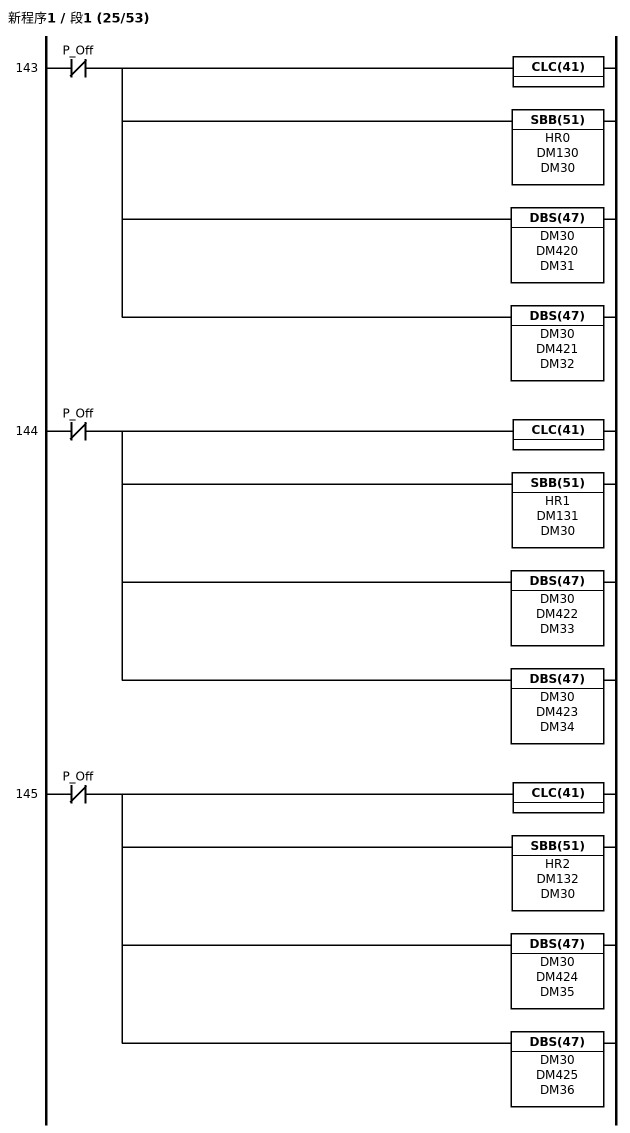
; [picture p24: 新程序1 / 段1, rungs 143-145]
; rung 143
LDNOT P_Off
CLC(41)
SBB(51) HR0 DM130 DM30
DBS(47) DM30 DM420 DM31
DBS(47) DM30 DM421 DM32
; rung 144
LDNOT P_Off
CLC(41)
SBB(51) HR1 DM131 DM30
DBS(47) DM30 DM422 DM33
DBS(47) DM30 DM423 DM34
; rung 145
LDNOT P_Off
CLC(41)
SBB(51) HR2 DM132 DM30
DBS(47) DM30 DM424 DM35
DBS(47) DM30 DM425 DM36

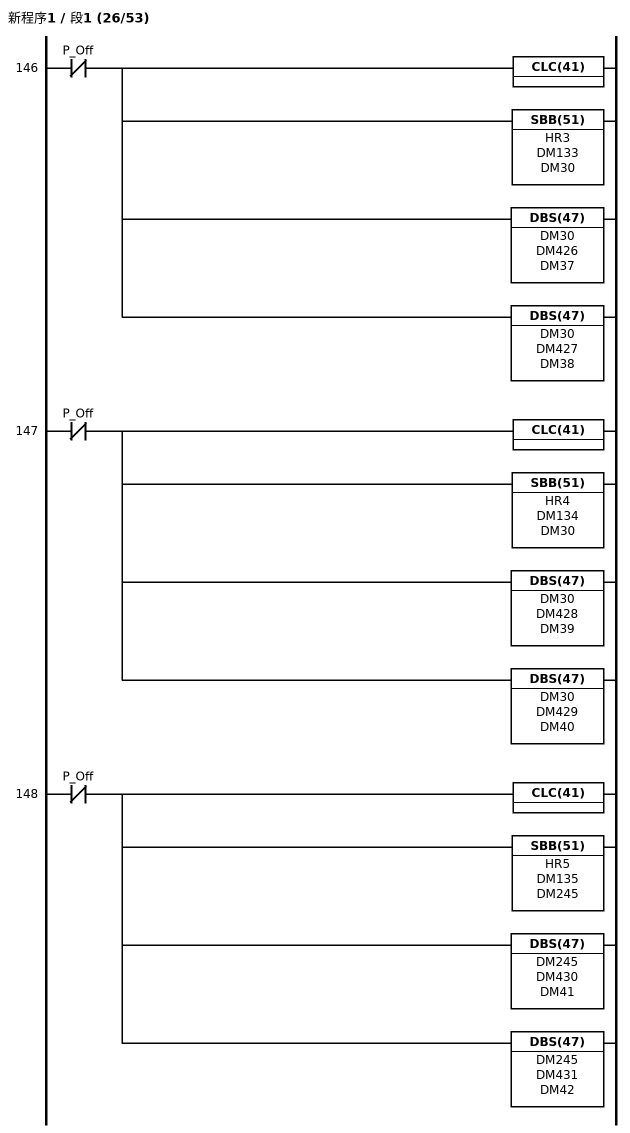
; rung 146
LDNOT P_Off
CLC(41)
SBB(51) HR3 DM133 DM30
DBS(47) DM30 DM426 DM37
DBS(47) DM30 DM427 DM38
; rung 147
LDNOT P_Off
CLC(41)
SBB(51) HR4 DM134 DM30
DBS(47) DM30 DM428 DM39
DBS(47) DM30 DM429 DM40
; rung 148
LDNOT P_Off
CLC(41)
SBB(51) HR5 DM135 DM245
DBS(47) DM245 DM430 DM41
DBS(47) DM245 DM431 DM42

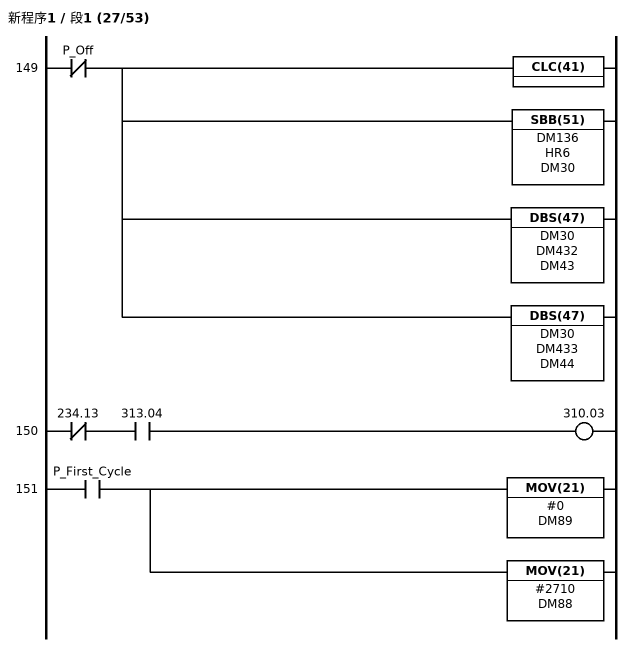
; rung 149
LDNOT P_Off
CLC(41)
SBB(51) DM136 HR6 DM30
DBS(47) DM30 DM432 DM43
DBS(47) DM30 DM433 DM44
; rung 150
LDNOT 234.13
AND 313.04
OUT 310.03
; rung 151
LD P_First_Cycle
MOV(21) #0 DM89
MOV(21) #2710 DM88

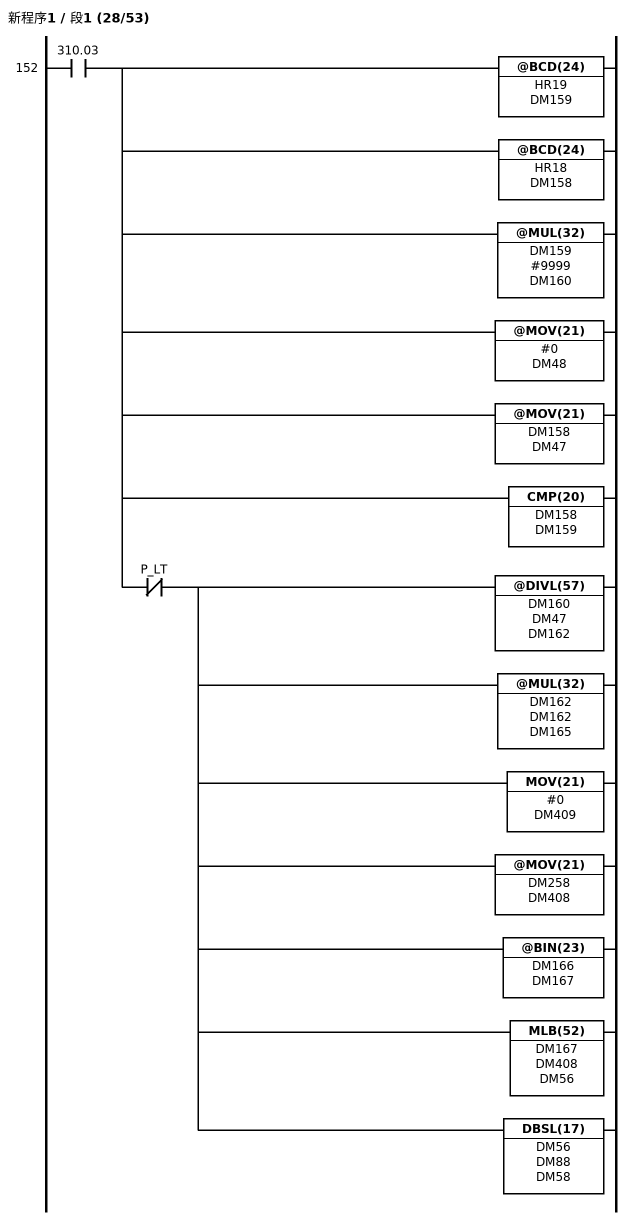
; rung 152
LD 310.03
@BCD(24) HR19 DM159
@BCD(24) HR18 DM158
@MUL(32) DM159 #9999 DM160
@MOV(21) #0 DM48
@MOV(21) DM158 DM47
CMP(20) DM158 DM159
ANDNOT P_LT
@DIVL(57) DM160 DM47 DM162
@MUL(32) DM162 DM162 DM165
MOV(21) #0 DM409
@MOV(21) DM258 DM408
@BIN(23) DM166 DM167
MLB(52) DM167 DM408 DM56
DBSL(17) DM56 DM88 DM58

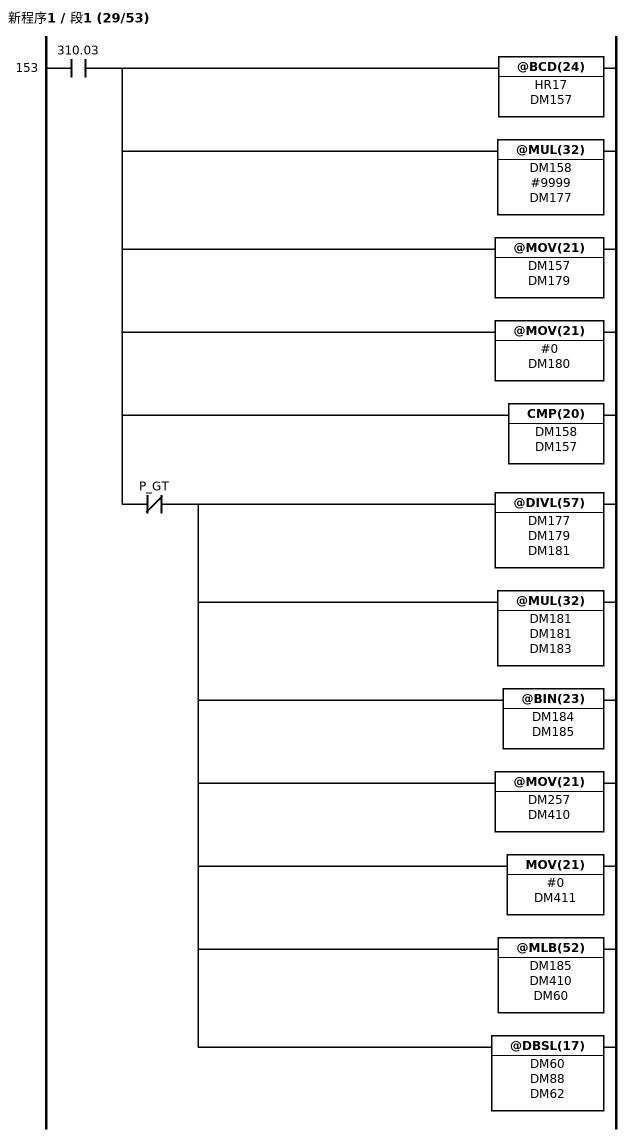
; rung 153
LD 310.03
@BCD(24) HR17 DM157
@MUL(32) DM158 #9999 DM177
@MOV(21) DM157 DM179
@MOV(21) #0 DM180
CMP(20) DM158 DM157
ANDNOT P_GT
@DIVL(57) DM177 DM179 DM181
@MUL(32) DM181 DM181 DM183
@BIN(23) DM184 DM185
@MOV(21) DM257 DM410
MOV(21) #0 DM411
@MLB(52) DM185 DM410 DM60
@DBSL(17) DM60 DM88 DM62

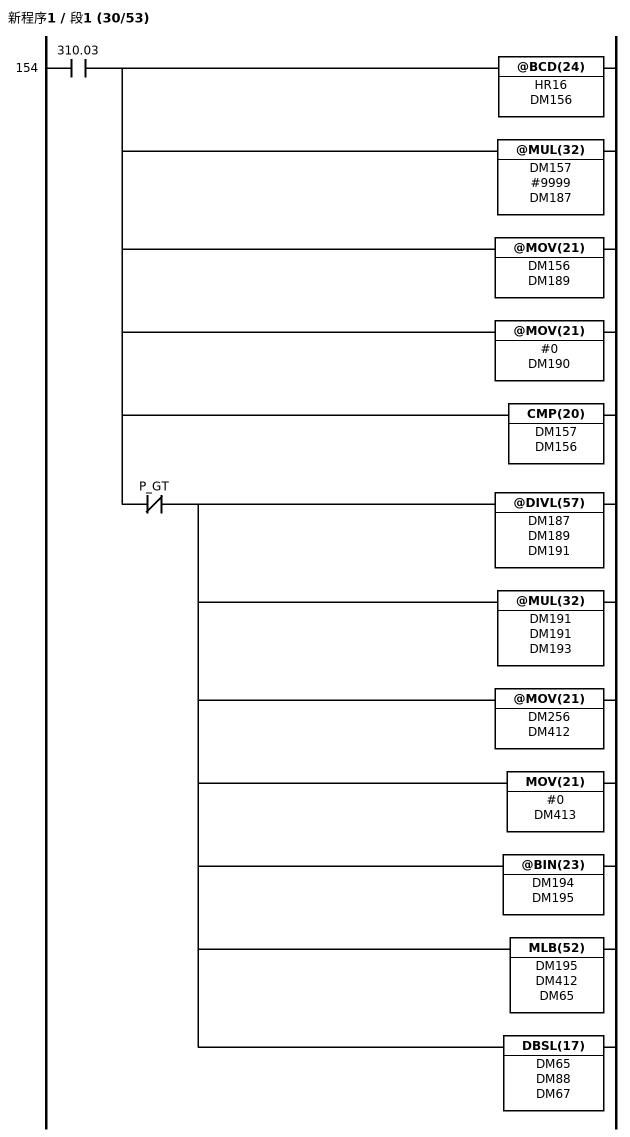
; rung 154
LD 310.03
@BCD(24) HR16 DM156
@MUL(32) DM157 #9999 DM187
@MOV(21) DM156 DM189
@MOV(21) #0 DM190
CMP(20) DM157 DM156
ANDNOT P_GT
@DIVL(57) DM187 DM189 DM191
@MUL(32) DM191 DM191 DM193
@MOV(21) DM256 DM412
MOV(21) #0 DM413
@BIN(23) DM194 DM195
MLB(52) DM195 DM412 DM65
DBSL(17) DM65 DM88 DM67

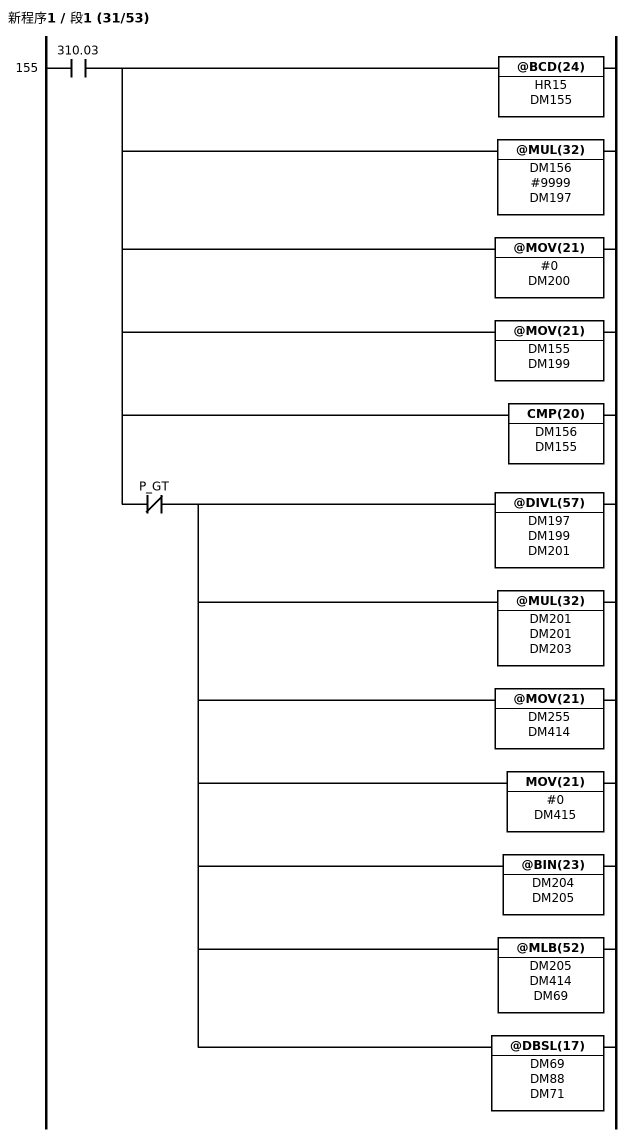
; rung 155
LD 310.03
@BCD(24) HR15 DM155
@MUL(32) DM156 #9999 DM197
@MOV(21) #0 DM200
@MOV(21) DM155 DM199
CMP(20) DM156 DM155
ANDNOT P_GT
@DIVL(57) DM197 DM199 DM201
@MUL(32) DM201 DM201 DM203
@MOV(21) DM255 DM414
MOV(21) #0 DM415
@BIN(23) DM204 DM205
@MLB(52) DM205 DM414 DM69
@DBSL(17) DM69 DM88 DM71

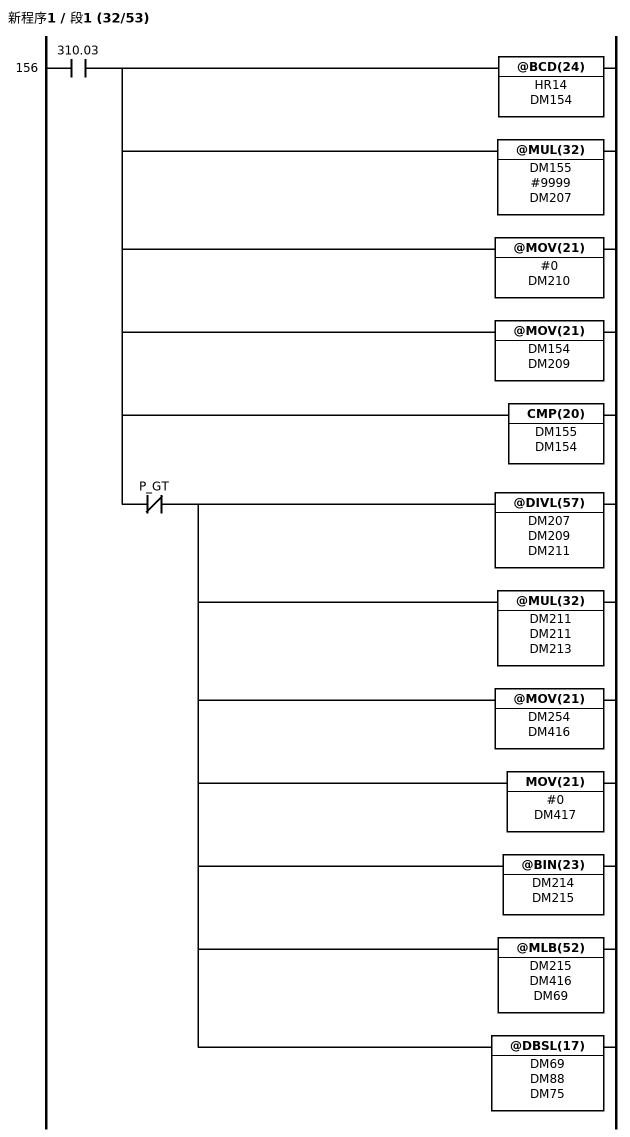
; rung 156
LD 310.03
@BCD(24) HR14 DM154
@MUL(32) DM155 #9999 DM207
@MOV(21) #0 DM210
@MOV(21) DM154 DM209
CMP(20) DM155 DM154
ANDNOT P_GT
@DIVL(57) DM207 DM209 DM211
@MUL(32) DM211 DM211 DM213
@MOV(21) DM254 DM416
MOV(21) #0 DM417
@BIN(23) DM214 DM215
@MLB(52) DM215 DM416 DM69
@DBSL(17) DM69 DM88 DM75

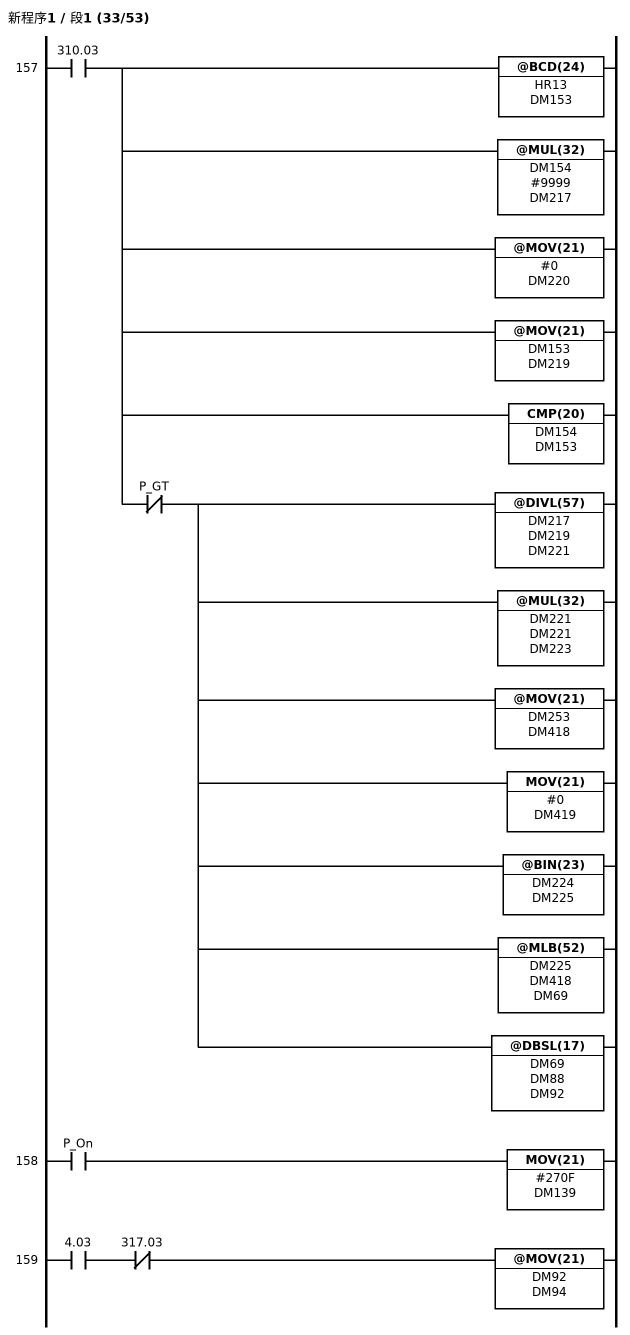
; rung 157
LD 310.03
@BCD(24) HR13 DM153
@MUL(32) DM154 #9999 DM217
@MOV(21) #0 DM220
@MOV(21) DM153 DM219
CMP(20) DM154 DM153
ANDNOT P_GT
@DIVL(57) DM217 DM219 DM221
@MUL(32) DM221 DM221 DM223
@MOV(21) DM253 DM418
MOV(21) #0 DM419
@BIN(23) DM224 DM225
@MLB(52) DM225 DM418 DM69
@DBSL(17) DM69 DM88 DM92
; rung 158
LD P_On
MOV(21) #270F DM139
; rung 159
LD 4.03
ANDNOT 317.03
@MOV(21) DM92 DM94

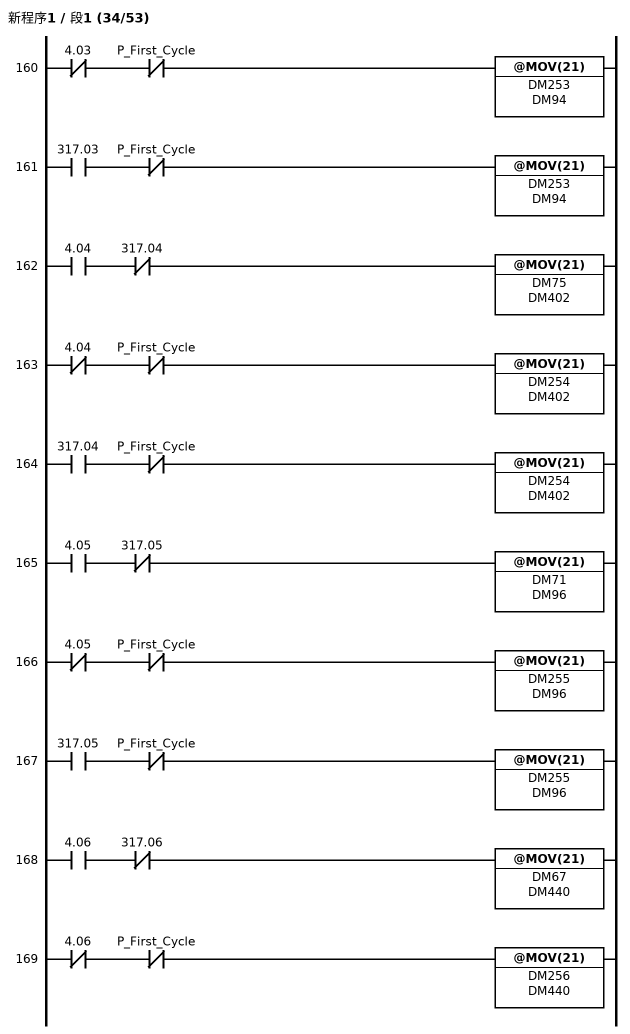
; rung 160
LDNOT 4.03
ANDNOT P_First_Cycle
@MOV(21) DM253 DM94
; rung 161
LD 317.03
ANDNOT P_First_Cycle
@MOV(21) DM253 DM94
; rung 162
LD 4.04
ANDNOT 317.04
@MOV(21) DM75 DM402
; rung 163
LDNOT 4.04
ANDNOT P_First_Cycle
@MOV(21) DM254 DM402
; rung 164
LD 317.04
ANDNOT P_First_Cycle
@MOV(21) DM254 DM402
; rung 165
LD 4.05
ANDNOT 317.05
@MOV(21) DM71 DM96
; rung 166
LDNOT 4.05
ANDNOT P_First_Cycle
@MOV(21) DM255 DM96
; rung 167
LD 317.05
ANDNOT P_First_Cycle
@MOV(21) DM255 DM96
; rung 168
LD 4.06
ANDNOT 317.06
@MOV(21) DM67 DM440
; rung 169
LDNOT 4.06
ANDNOT P_First_Cycle
@MOV(21) DM256 DM440

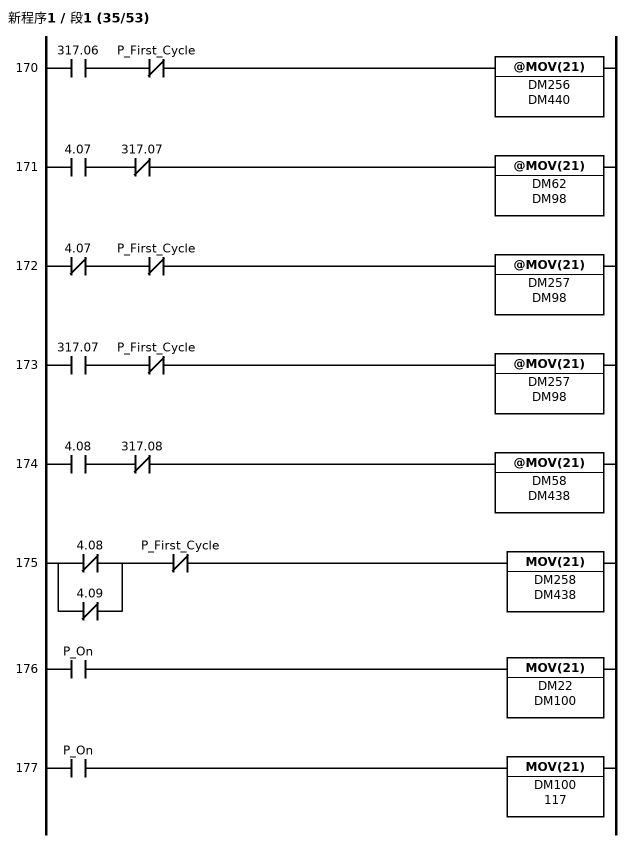
; rung 170
LD 317.06
ANDNOT P_First_Cycle
@MOV(21) DM256 DM440
; rung 171
LD 4.07
ANDNOT 317.07
@MOV(21) DM62 DM98
; rung 172
LDNOT 4.07
ANDNOT P_First_Cycle
@MOV(21) DM257 DM98
; rung 173
LD 317.07
ANDNOT P_First_Cycle
@MOV(21) DM257 DM98
; rung 174
LD 4.08
ANDNOT 317.08
@MOV(21) DM58 DM438
; rung 175
LDNOT 4.08
ORNOT 4.09
ANDNOT P_First_Cycle
MOV(21) DM258 DM438
; rung 176
LD P_On
MOV(21) DM22 DM100
; rung 177
LD P_On
MOV(21) DM100 117

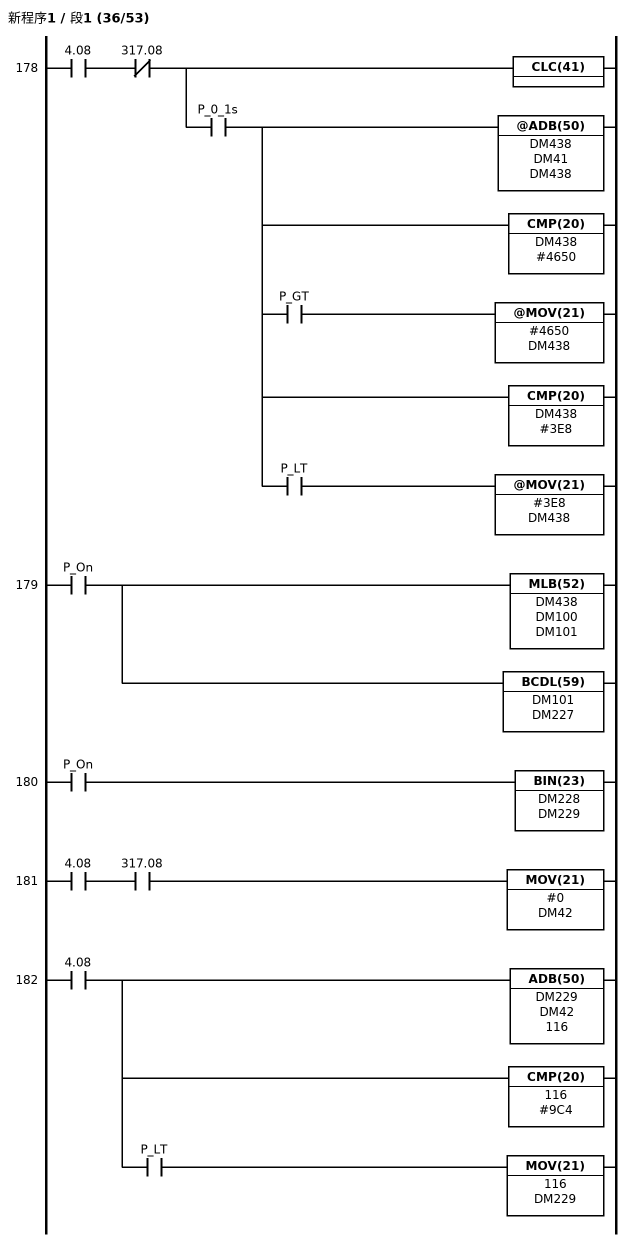
; rung 178
LD 4.08
ANDNOT 317.08
CLC(41)
AND P_0_1s
OUT TR0
@ADB(50) DM438 DM41 DM438
CMP(20) DM438 #4650
AND P_GT
@MOV(21) #4650 DM438
LD TR0
CMP(20) DM438 #3E8
AND P_LT
@MOV(21) #3E8 DM438
; rung 179
LD P_On
MLB(52) DM438 DM100 DM101
BCDL(59) DM101 DM227
; rung 180
LD P_On
BIN(23) DM228 DM229
; rung 181
LD 4.08
AND 317.08
MOV(21) #0 DM42
; rung 182
LD 4.08
ADB(50) DM229 DM42 116
CMP(20) 116 #9C4
AND P_LT
MOV(21) 116 DM229

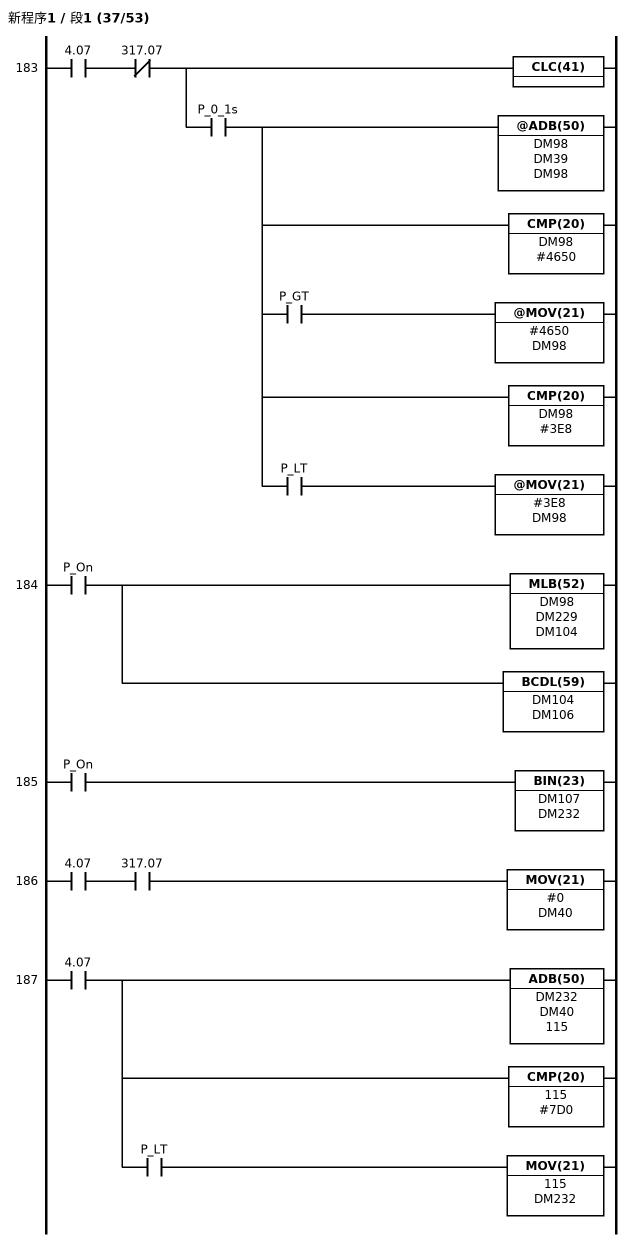
; rung 183
LD 4.07
ANDNOT 317.07
CLC(41)
AND P_0_1s
OUT TR0
@ADB(50) DM98 DM39 DM98
CMP(20) DM98 #4650
AND P_GT
@MOV(21) #4650 DM98
LD TR0
CMP(20) DM98 #3E8
AND P_LT
@MOV(21) #3E8 DM98
; rung 184
LD P_On
MLB(52) DM98 DM229 DM104
BCDL(59) DM104 DM106
; rung 185
LD P_On
BIN(23) DM107 DM232
; rung 186
LD 4.07
AND 317.07
MOV(21) #0 DM40
; rung 187
LD 4.07
ADB(50) DM232 DM40 115
CMP(20) 115 #7D0
AND P_LT
MOV(21) 115 DM232

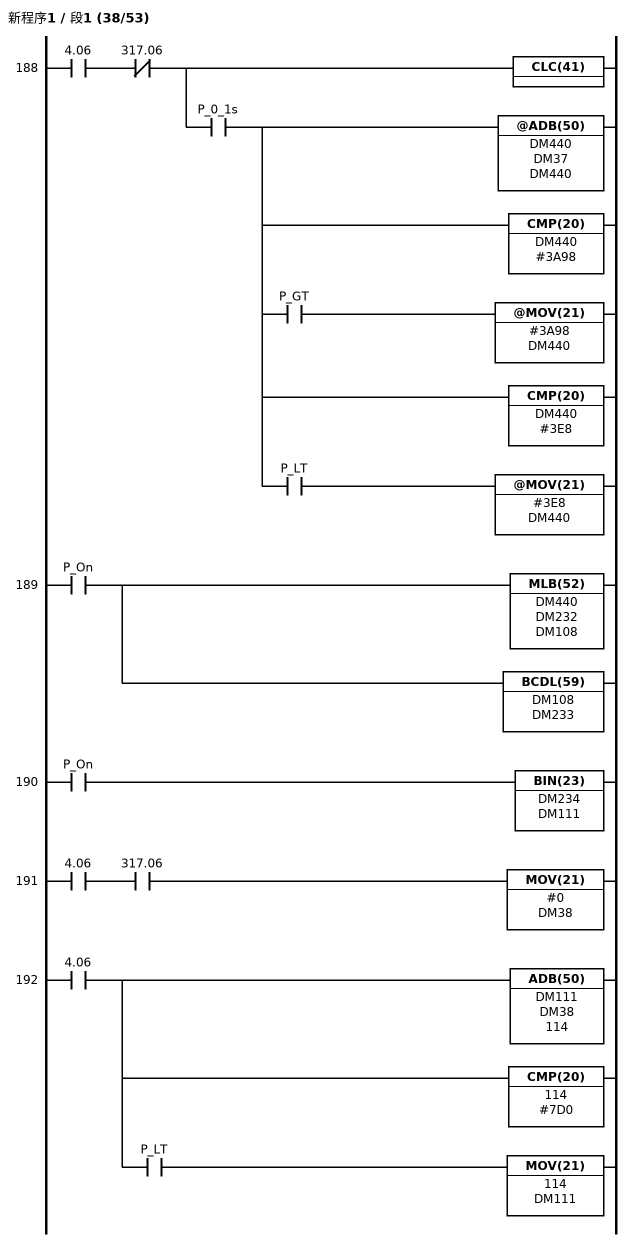
; rung 188
LD 4.06
ANDNOT 317.06
CLC(41)
AND P_0_1s
OUT TR0
@ADB(50) DM440 DM37 DM440
CMP(20) DM440 #3A98
AND P_GT
@MOV(21) #3A98 DM440
LD TR0
CMP(20) DM440 #3E8
AND P_LT
@MOV(21) #3E8 DM440
; rung 189
LD P_On
MLB(52) DM440 DM232 DM108
BCDL(59) DM108 DM233
; rung 190
LD P_On
BIN(23) DM234 DM111
; rung 191
LD 4.06
AND 317.06
MOV(21) #0 DM38
; rung 192
LD 4.06
ADB(50) DM111 DM38 114
CMP(20) 114 #7D0
AND P_LT
MOV(21) 114 DM111

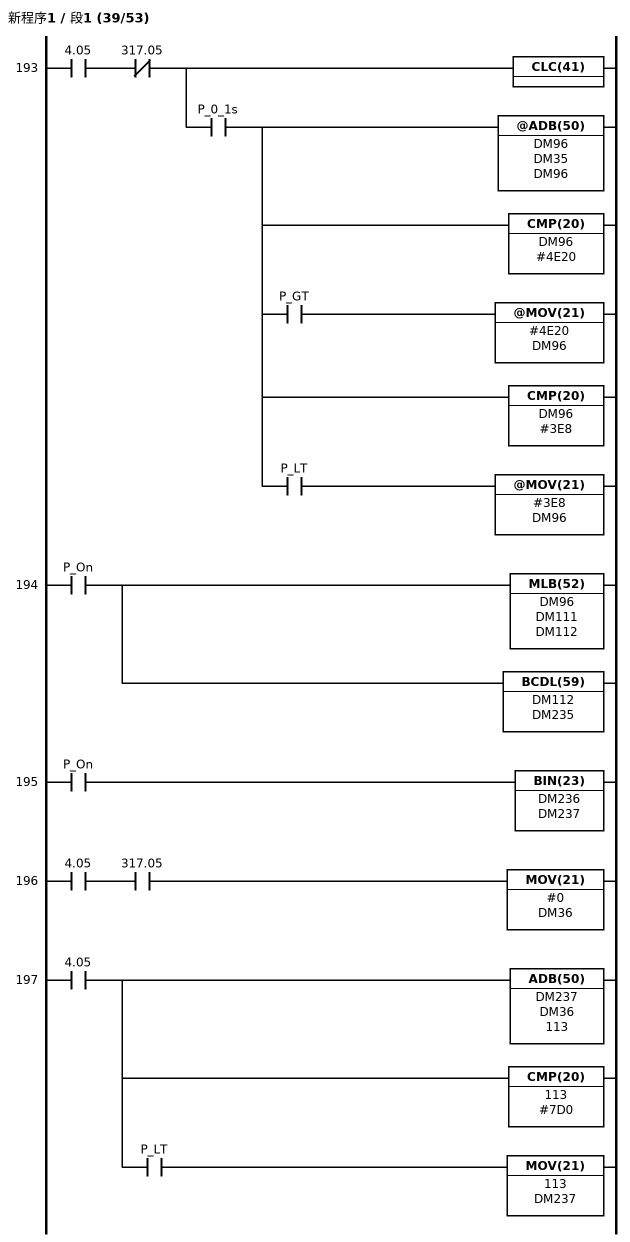
; rung 193
LD 4.05
ANDNOT 317.05
CLC(41)
AND P_0_1s
OUT TR0
@ADB(50) DM96 DM35 DM96
CMP(20) DM96 #4E20
AND P_GT
@MOV(21) #4E20 DM96
LD TR0
CMP(20) DM96 #3E8
AND P_LT
@MOV(21) #3E8 DM96
; rung 194
LD P_On
MLB(52) DM96 DM111 DM112
BCDL(59) DM112 DM235
; rung 195
LD P_On
BIN(23) DM236 DM237
; rung 196
LD 4.05
AND 317.05
MOV(21) #0 DM36
; rung 197
LD 4.05
ADB(50) DM237 DM36 113
CMP(20) 113 #7D0
AND P_LT
MOV(21) 113 DM237

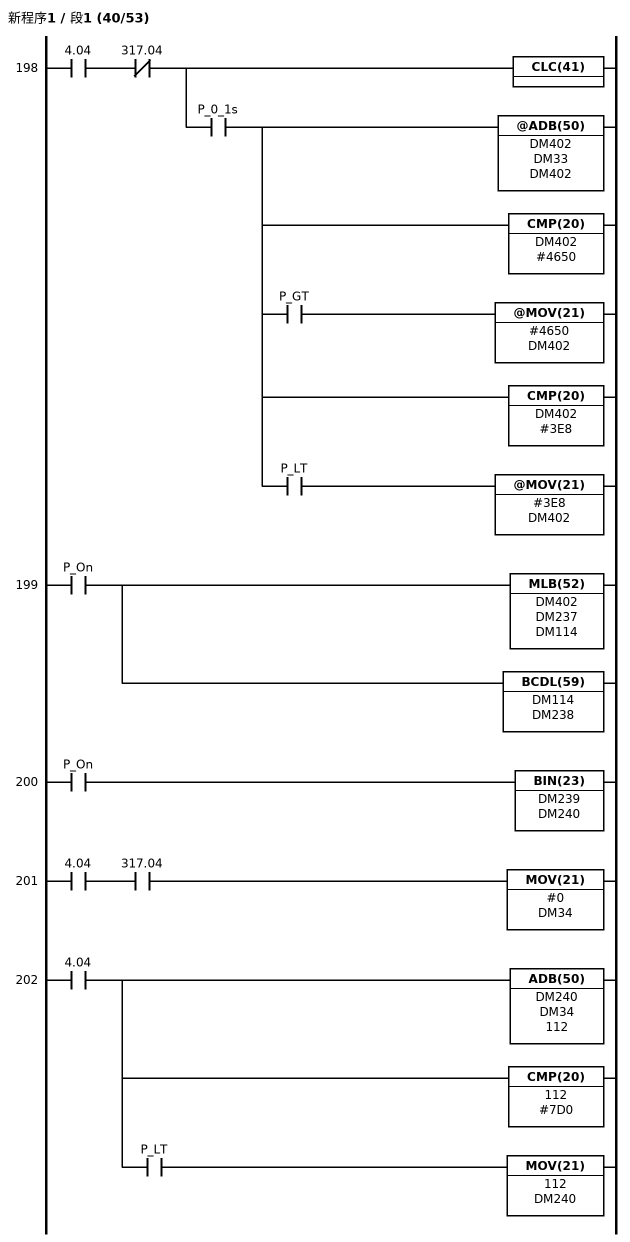
; rung 198
LD 4.04
ANDNOT 317.04
CLC(41)
AND P_0_1s
OUT TR0
@ADB(50) DM402 DM33 DM402
CMP(20) DM402 #4650
AND P_GT
@MOV(21) #4650 DM402
LD TR0
CMP(20) DM402 #3E8
AND P_LT
@MOV(21) #3E8 DM402
; rung 199
LD P_On
MLB(52) DM402 DM237 DM114
BCDL(59) DM114 DM238
; rung 200
LD P_On
BIN(23) DM239 DM240
; rung 201
LD 4.04
AND 317.04
MOV(21) #0 DM34
; rung 202
LD 4.04
ADB(50) DM240 DM34 112
CMP(20) 112 #7D0
AND P_LT
MOV(21) 112 DM240

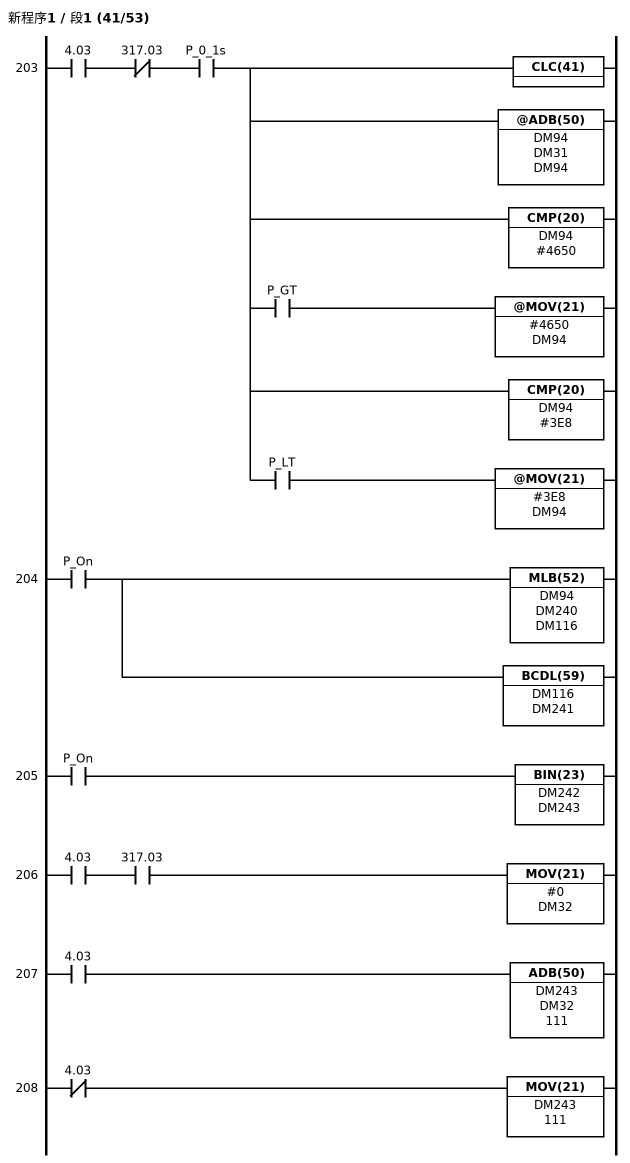
; rung 203
LD 4.03
ANDNOT 317.03
AND P_0_1s
OUT TR0
CLC(41)
@ADB(50) DM94 DM31 DM94
CMP(20) DM94 #4650
AND P_GT
@MOV(21) #4650 DM94
LD TR0
CMP(20) DM94 #3E8
AND P_LT
@MOV(21) #3E8 DM94
; rung 204
LD P_On
MLB(52) DM94 DM240 DM116
BCDL(59) DM116 DM241
; rung 205
LD P_On
BIN(23) DM242 DM243
; rung 206
LD 4.03
AND 317.03
MOV(21) #0 DM32
; rung 207
LD 4.03
ADB(50) DM243 DM32 111
; rung 208
LDNOT 4.03
MOV(21) DM243 111

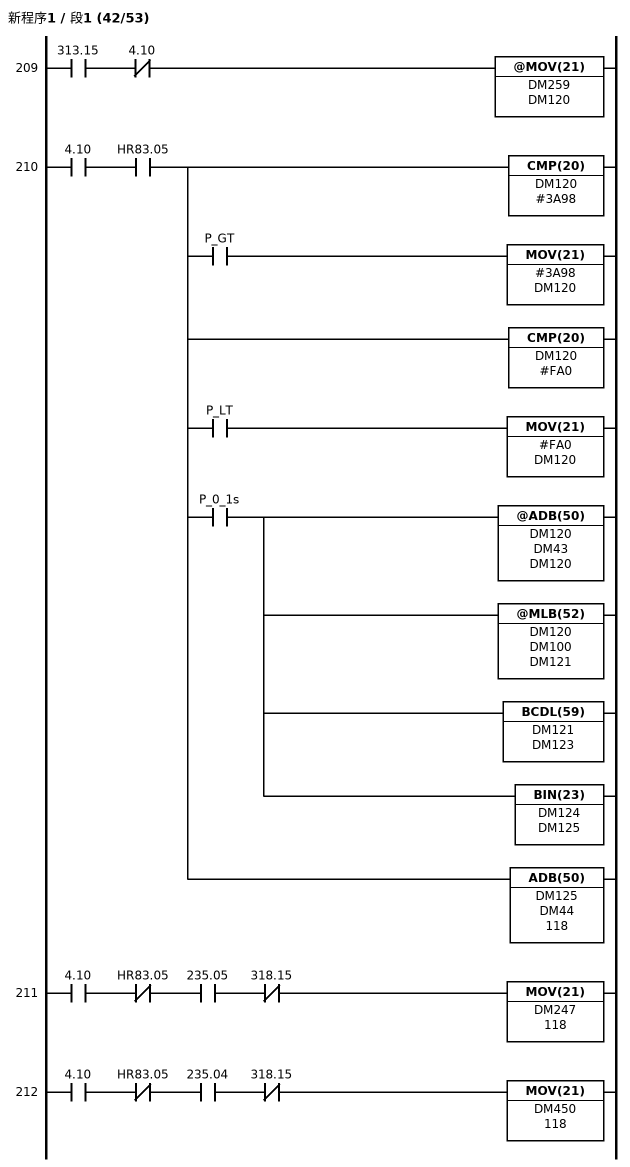
; rung 209
LD 313.15
ANDNOT 4.10
@MOV(21) DM259 DM120
; rung 210
LD 4.10
AND HR83.05
OUT TR0
CMP(20) DM120 #3A98
AND P_GT
MOV(21) #3A98 DM120
LD TR0
CMP(20) DM120 #FA0
AND P_LT
MOV(21) #FA0 DM120
LD TR0
AND P_0_1s
@ADB(50) DM120 DM43 DM120
@MLB(52) DM120 DM100 DM121
BCDL(59) DM121 DM123
BIN(23) DM124 DM125
LD TR0
ADB(50) DM125 DM44 118
; rung 211
LD 4.10
ANDNOT HR83.05
AND 235.05
ANDNOT 318.15
MOV(21) DM247 118
; rung 212
LD 4.10
ANDNOT HR83.05
AND 235.04
ANDNOT 318.15
MOV(21) DM450 118

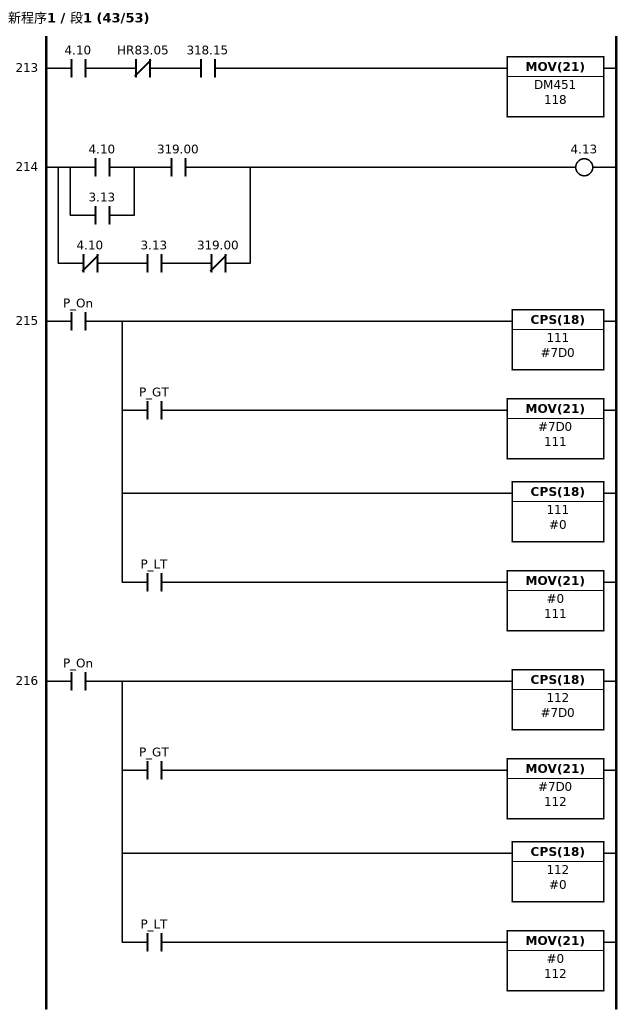
; rung 213
LD 4.10
ANDNOT HR83.05
AND 318.15
MOV(21) DM451 118
; rung 214
LD 4.10
OR 3.13
AND 319.00
LDNOT 4.10
AND 3.13
ANDNOT 319.00
ORLD
OUT 4.13
; rung 215
LD P_On
OUT TR0
CPS(18) 111 #7D0
AND P_GT
MOV(21) #7D0 111
LD TR0
CPS(18) 111 #0
AND P_LT
MOV(21) #0 111
; rung 216
LD P_On
OUT TR0
CPS(18) 112 #7D0
AND P_GT
MOV(21) #7D0 112
LD TR0
CPS(18) 112 #0
AND P_LT
MOV(21) #0 112

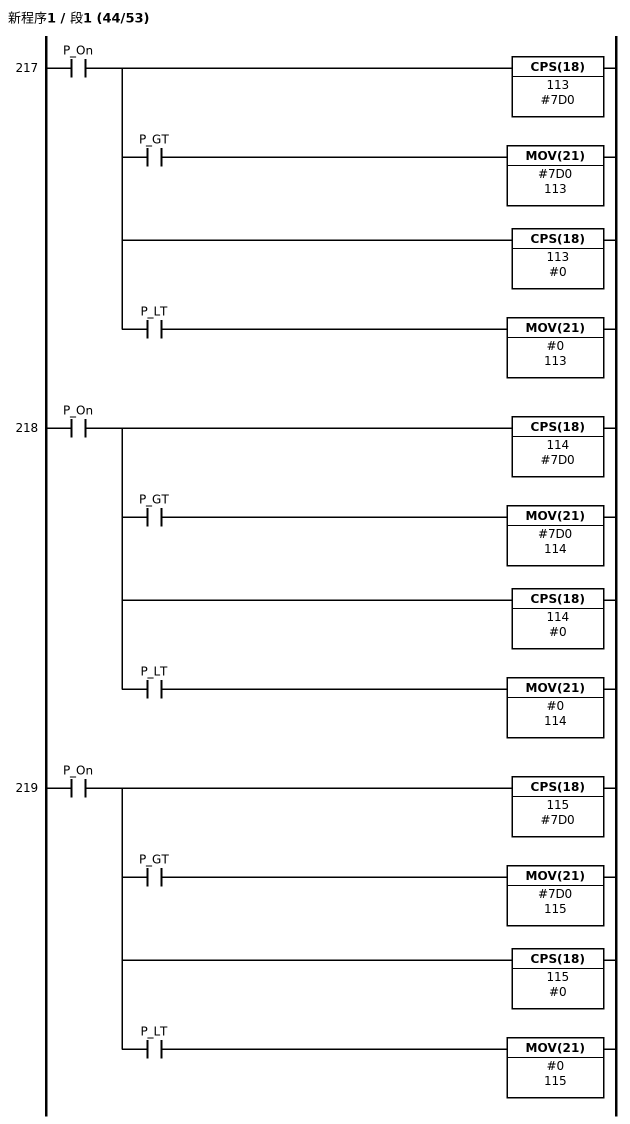
; rung 217
LD P_On
OUT TR0
CPS(18) 113 #7D0
AND P_GT
MOV(21) #7D0 113
LD TR0
CPS(18) 113 #0
AND P_LT
MOV(21) #0 113
; rung 218
LD P_On
OUT TR0
CPS(18) 114 #7D0
AND P_GT
MOV(21) #7D0 114
LD TR0
CPS(18) 114 #0
AND P_LT
MOV(21) #0 114
; rung 219
LD P_On
OUT TR0
CPS(18) 115 #7D0
AND P_GT
MOV(21) #7D0 115
LD TR0
CPS(18) 115 #0
AND P_LT
MOV(21) #0 115

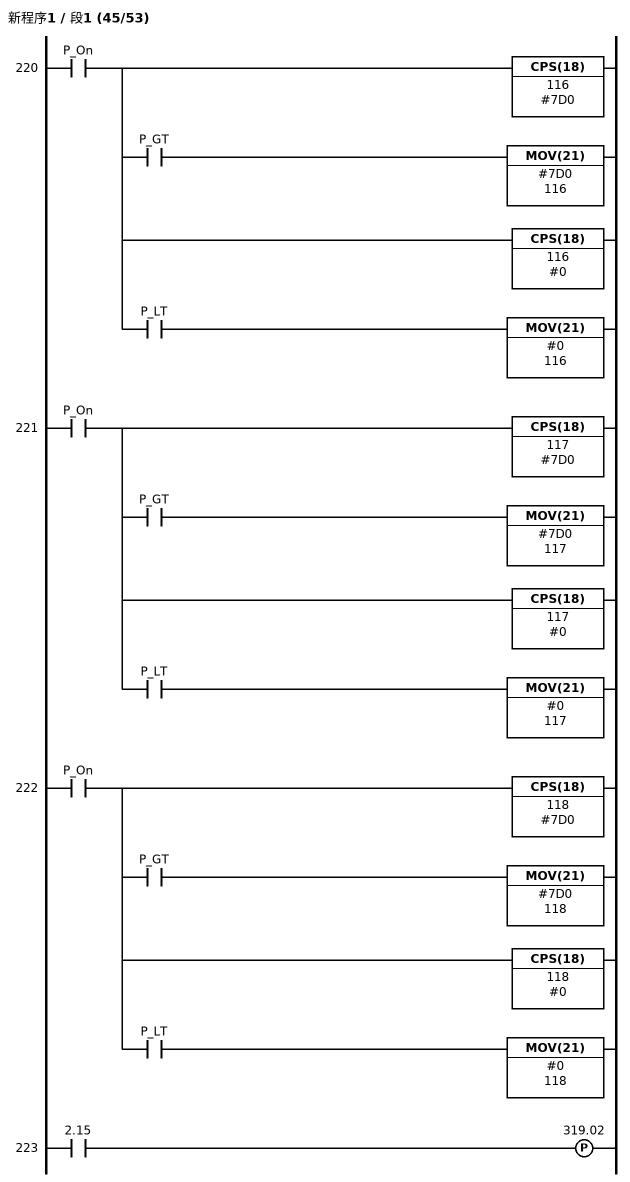
; rung 220
LD P_On
OUT TR0
CPS(18) 116 #7D0
AND P_GT
MOV(21) #7D0 116
LD TR0
CPS(18) 116 #0
AND P_LT
MOV(21) #0 116
; rung 221
LD P_On
OUT TR0
CPS(18) 117 #7D0
AND P_GT
MOV(21) #7D0 117
LD TR0
CPS(18) 117 #0
AND P_LT
MOV(21) #0 117
; rung 222
LD P_On
OUT TR0
CPS(18) 118 #7D0
AND P_GT
MOV(21) #7D0 118
LD TR0
CPS(18) 118 #0
AND P_LT
MOV(21) #0 118
; rung 223
LD 2.15
DIFU(13) 319.02

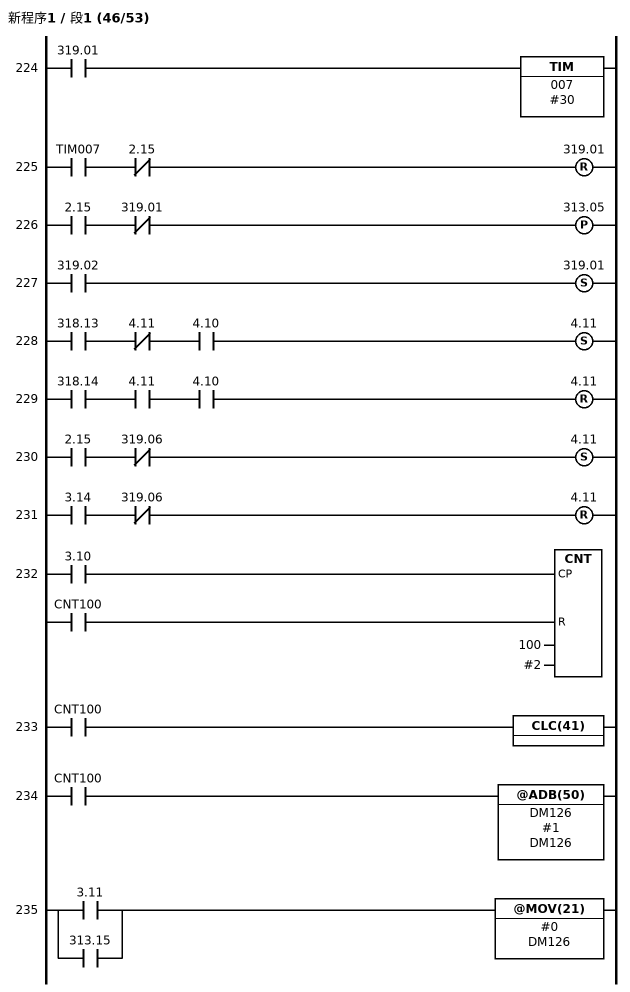
; rung 224
LD 319.01
TIM 007 #30
; rung 225
LD TIM007
ANDNOT 2.15
RSET 319.01
; rung 226
LD 2.15
ANDNOT 319.01
DIFU(13) 313.05
; rung 227
LD 319.02
SET 319.01
; rung 228
LD 318.13
ANDNOT 4.11
AND 4.10
SET 4.11
; rung 229
LD 318.14
AND 4.11
AND 4.10
RSET 4.11
; rung 230
LD 2.15
ANDNOT 319.06
SET 4.11
; rung 231
LD 3.14
ANDNOT 319.06
RSET 4.11
; rung 232
LD 3.10
LD CNT100
CNT 100 #2
; rung 233
LD CNT100
CLC(41)
; rung 234
LD CNT100
@ADB(50) DM126 #1 DM126
; rung 235
LD 3.11
OR 313.15
@MOV(21) #0 DM126

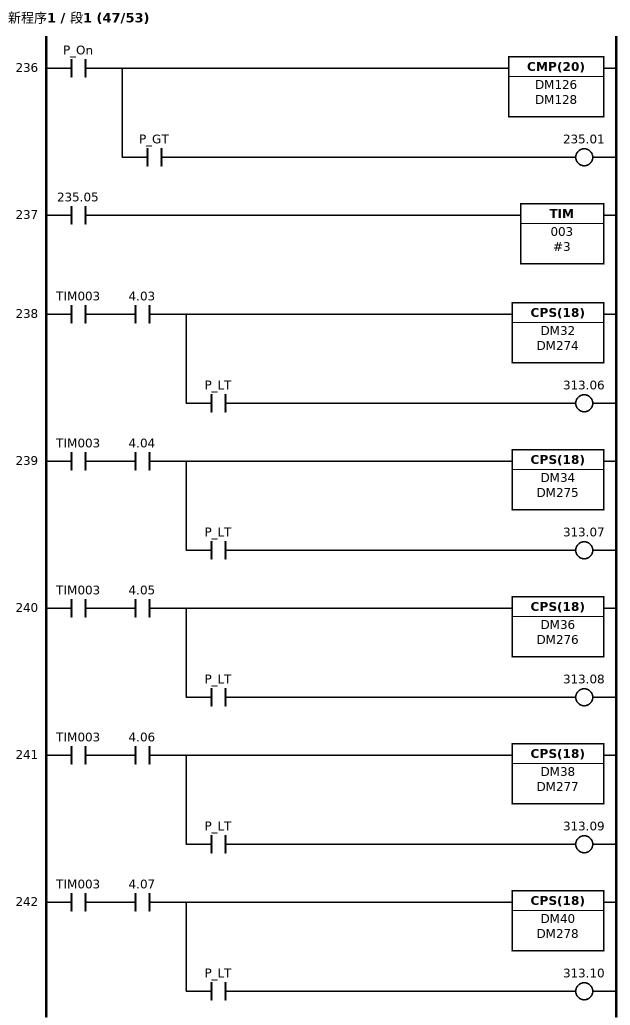
; rung 236
LD P_On
CMP(20) DM126 DM128
AND P_GT
OUT 235.01
; rung 237
LD 235.05
TIM 003 #3
; rung 238
LD TIM003
AND 4.03
CPS(18) DM32 DM274
AND P_LT
OUT 313.06
; rung 239
LD TIM003
AND 4.04
CPS(18) DM34 DM275
AND P_LT
OUT 313.07
; rung 240
LD TIM003
AND 4.05
CPS(18) DM36 DM276
AND P_LT
OUT 313.08
; rung 241
LD TIM003
AND 4.06
CPS(18) DM38 DM277
AND P_LT
OUT 313.09
; rung 242
LD TIM003
AND 4.07
CPS(18) DM40 DM278
AND P_LT
OUT 313.10

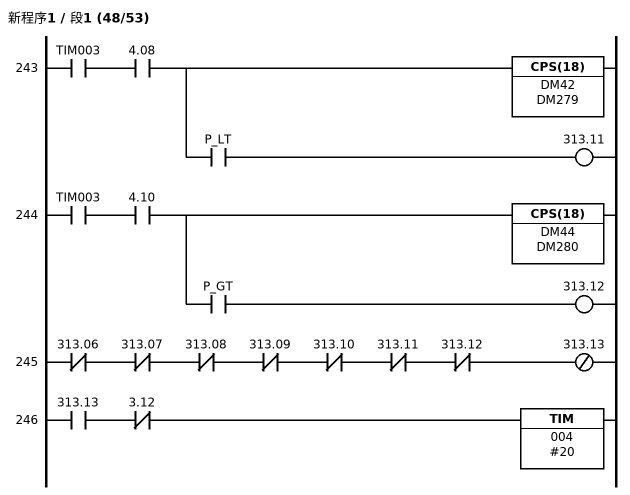
; rung 243
LD TIM003
AND 4.08
CPS(18) DM42 DM279
AND P_LT
OUT 313.11
; rung 244
LD TIM003
AND 4.10
CPS(18) DM44 DM280
AND P_GT
OUT 313.12
; rung 245
LDNOT 313.06
ANDNOT 313.07
ANDNOT 313.08
ANDNOT 313.09
ANDNOT 313.10
ANDNOT 313.11
ANDNOT 313.12
OUTNOT 313.13
; rung 246
LD 313.13
ANDNOT 3.12
TIM 004 #20

